PROGRAM IO_OP10_PANEL
VAR
	OP10_MP_16DI_MODULE_1 AT %I* : WORD;
	OP10_MP_16DI_MODULE_2 AT %I* : WORD;
	OP10_MP_16DI_MODULE_3 AT %I* : WORD;
	OP10_MP_16DI_MODULE_4 AT %I* : WORD;
	OP10_MP_16DI_MODULE_5 AT %I* : WORD;
	OP10_MP_16DI_MODULE_6 AT %I* : WORD;
	
	OP10_MP_16DO_MODULE_1 AT %Q* : WORD;
	OP10_MP_16DO_MODULE_2 AT %Q* : WORD;
	OP10_MP_16DO_MODULE_3 AT %Q* : WORD;
	OP10_MP_16DO_MODULE_4 AT %Q* : WORD;
	OP10_MP_16DO_MODULE_5 AT %Q* : WORD;
	
	WORD_AS_BIT_0: WORD_AS_BIT;
	WORD_AS_BIT_1: WORD_AS_BIT;
	WORD_AS_BIT_2: WORD_AS_BIT;
	WORD_AS_BIT_3: WORD_AS_BIT;
	WORD_AS_BIT_4: WORD_AS_BIT;
	WORD_AS_BIT_5: WORD_AS_BIT;

	BIT_AS_WORD_0: BIT_AS_WORD;
	BIT_AS_WORD_1: BIT_AS_WORD;
	BIT_AS_WORD_2: BIT_AS_WORD;
	BIT_AS_WORD_3: BIT_AS_WORD;
	BIT_AS_WORD_4: BIT_AS_WORD;
	OP10_MP_Spare_byte: WORD;
END_VAR

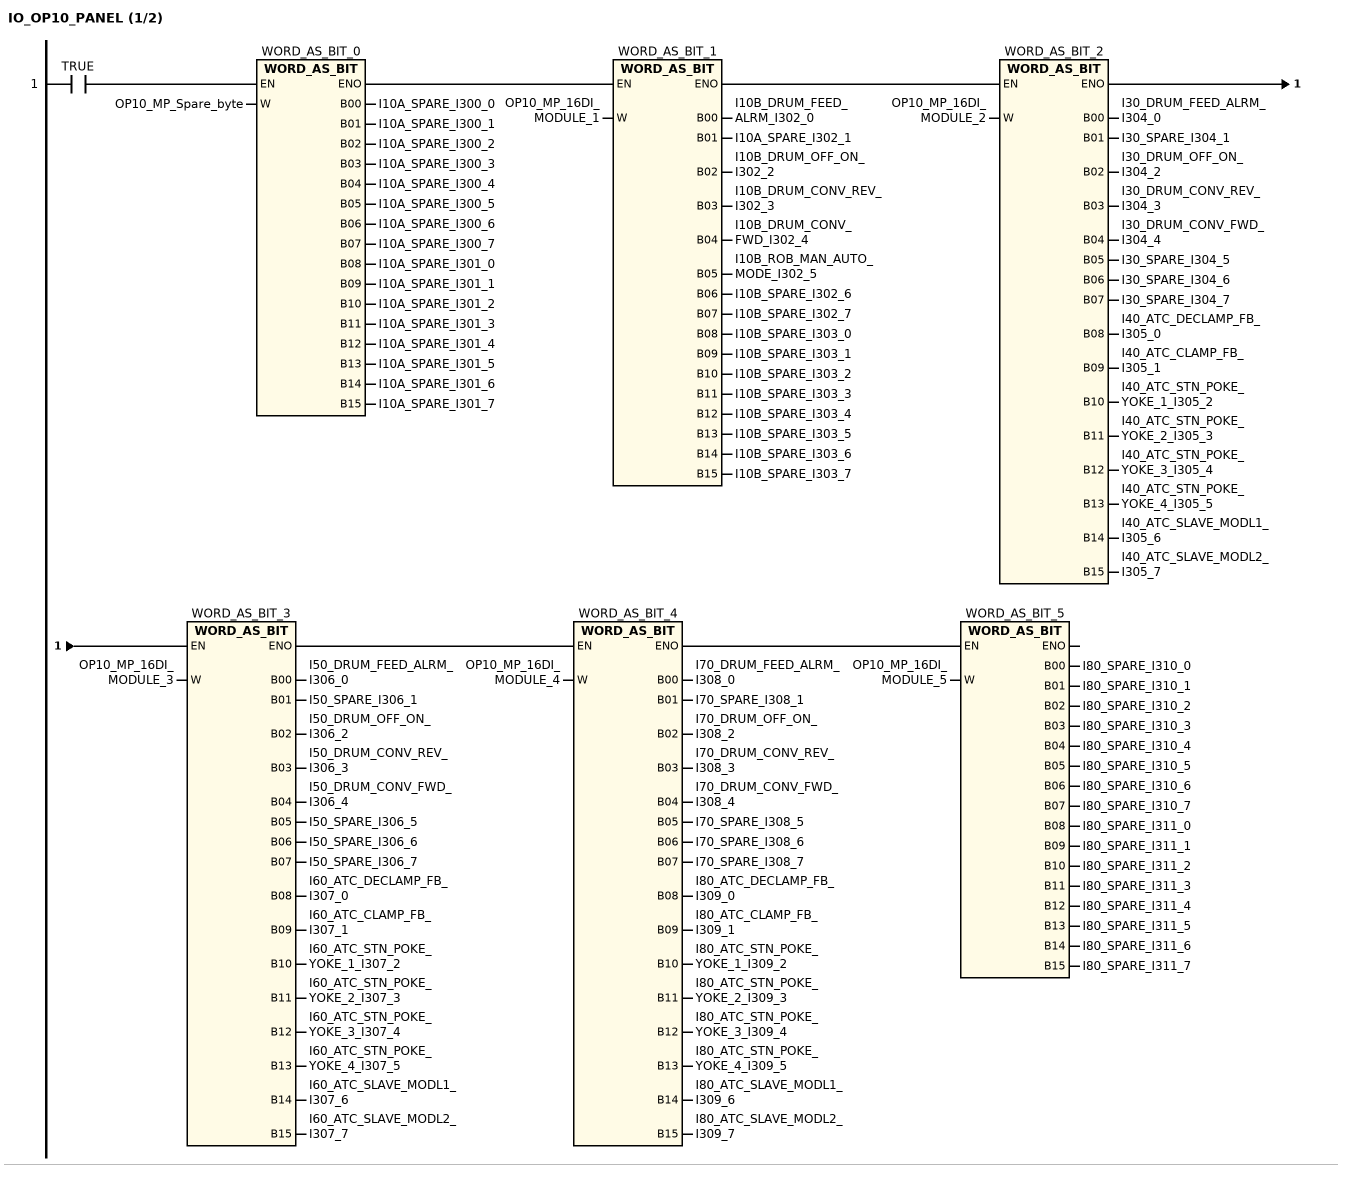
// NETWORK 1
WORD_AS_BIT_0(
    W := OP10_MP_Spare_byte,
    B00 => I10A_SPARE_I300_0,
    B01 => I10A_SPARE_I300_1,
    B02 => I10A_SPARE_I300_2,
    B03 => I10A_SPARE_I300_3,
    B04 => I10A_SPARE_I300_4,
    B05 => I10A_SPARE_I300_5,
    B06 => I10A_SPARE_I300_6,
    B07 => I10A_SPARE_I300_7,
    B08 => I10A_SPARE_I301_0,
    B09 => I10A_SPARE_I301_1,
    B10 => I10A_SPARE_I301_2,
    B11 => I10A_SPARE_I301_3,
    B12 => I10A_SPARE_I301_4,
    B13 => I10A_SPARE_I301_5,
    B14 => I10A_SPARE_I301_6,
    B15 => I10A_SPARE_I301_7); // WORD_AS_BIT
WORD_AS_BIT_1(
    W := OP10_MP_16DI_MODULE_1,
    B00 => I10B_DRUM_FEED_ALRM_I302_0,
    B01 => I10A_SPARE_I302_1,
    B02 => I10B_DRUM_OFF_ON_I302_2,
    B03 => I10B_DRUM_CONV_REV_I302_3,
    B04 => I10B_DRUM_CONV_FWD_I302_4,
    B05 => I10B_ROB_MAN_AUTO_MODE_I302_5,
    B06 => I10B_SPARE_I302_6,
    B07 => I10B_SPARE_I302_7,
    B08 => I10B_SPARE_I303_0,
    B09 => I10B_SPARE_I303_1,
    B10 => I10B_SPARE_I303_2,
    B11 => I10B_SPARE_I303_3,
    B12 => I10B_SPARE_I303_4,
    B13 => I10B_SPARE_I303_5,
    B14 => I10B_SPARE_I303_6,
    B15 => I10B_SPARE_I303_7); // WORD_AS_BIT
WORD_AS_BIT_2(
    W := OP10_MP_16DI_MODULE_2,
    B00 => I30_DRUM_FEED_ALRM_I304_0,
    B01 => I30_SPARE_I304_1,
    B02 => I30_DRUM_OFF_ON_I304_2,
    B03 => I30_DRUM_CONV_REV_I304_3,
    B04 => I30_DRUM_CONV_FWD_I304_4,
    B05 => I30_SPARE_I304_5,
    B06 => I30_SPARE_I304_6,
    B07 => I30_SPARE_I304_7,
    B08 => I40_ATC_DECLAMP_FB_I305_0,
    B09 => I40_ATC_CLAMP_FB_I305_1,
    B10 => I40_ATC_STN_POKE_YOKE_1_I305_2,
    B11 => I40_ATC_STN_POKE_YOKE_2_I305_3,
    B12 => I40_ATC_STN_POKE_YOKE_3_I305_4,
    B13 => I40_ATC_STN_POKE_YOKE_4_I305_5,
    B14 => I40_ATC_SLAVE_MODL1_I305_6,
    B15 => I40_ATC_SLAVE_MODL2_I305_7); // WORD_AS_BIT
WORD_AS_BIT_3(
    W := OP10_MP_16DI_MODULE_3,
    B00 => I50_DRUM_FEED_ALRM_I306_0,
    B01 => I50_SPARE_I306_1,
    B02 => I50_DRUM_OFF_ON_I306_2,
    B03 => I50_DRUM_CONV_REV_I306_3,
    B04 => I50_DRUM_CONV_FWD_I306_4,
    B05 => I50_SPARE_I306_5,
    B06 => I50_SPARE_I306_6,
    B07 => I50_SPARE_I306_7,
    B08 => I60_ATC_DECLAMP_FB_I307_0,
    B09 => I60_ATC_CLAMP_FB_I307_1,
    B10 => I60_ATC_STN_POKE_YOKE_1_I307_2,
    B11 => I60_ATC_STN_POKE_YOKE_2_I307_3,
    B12 => I60_ATC_STN_POKE_YOKE_3_I307_4,
    B13 => I60_ATC_STN_POKE_YOKE_4_I307_5,
    B14 => I60_ATC_SLAVE_MODL1_I307_6,
    B15 => I60_ATC_SLAVE_MODL2_I307_7); // WORD_AS_BIT
WORD_AS_BIT_4(
    W := OP10_MP_16DI_MODULE_4,
    B00 => I70_DRUM_FEED_ALRM_I308_0,
    B01 => I70_SPARE_I308_1,
    B02 => I70_DRUM_OFF_ON_I308_2,
    B03 => I70_DRUM_CONV_REV_I308_3,
    B04 => I70_DRUM_CONV_FWD_I308_4,
    B05 => I70_SPARE_I308_5,
    B06 => I70_SPARE_I308_6,
    B07 => I70_SPARE_I308_7,
    B08 => I80_ATC_DECLAMP_FB_I309_0,
    B09 => I80_ATC_CLAMP_FB_I309_1,
    B10 => I80_ATC_STN_POKE_YOKE_1_I309_2,
    B11 => I80_ATC_STN_POKE_YOKE_2_I309_3,
    B12 => I80_ATC_STN_POKE_YOKE_3_I309_4,
    B13 => I80_ATC_STN_POKE_YOKE_4_I309_5,
    B14 => I80_ATC_SLAVE_MODL1_I309_6,
    B15 => I80_ATC_SLAVE_MODL2_I309_7); // WORD_AS_BIT
WORD_AS_BIT_5(
    W := OP10_MP_16DI_MODULE_5,
    B00 => I80_SPARE_I310_0,
    B01 => I80_SPARE_I310_1,
    B02 => I80_SPARE_I310_2,
    B03 => I80_SPARE_I310_3,
    B04 => I80_SPARE_I310_4,
    B05 => I80_SPARE_I310_5,
    B06 => I80_SPARE_I310_6,
    B07 => I80_SPARE_I310_7,
    B08 => I80_SPARE_I311_0,
    B09 => I80_SPARE_I311_1,
    B10 => I80_SPARE_I311_2,
    B11 => I80_SPARE_I311_3,
    B12 => I80_SPARE_I311_4,
    B13 => I80_SPARE_I311_5,
    B14 => I80_SPARE_I311_6,
    B15 => I80_SPARE_I311_7); // WORD_AS_BIT

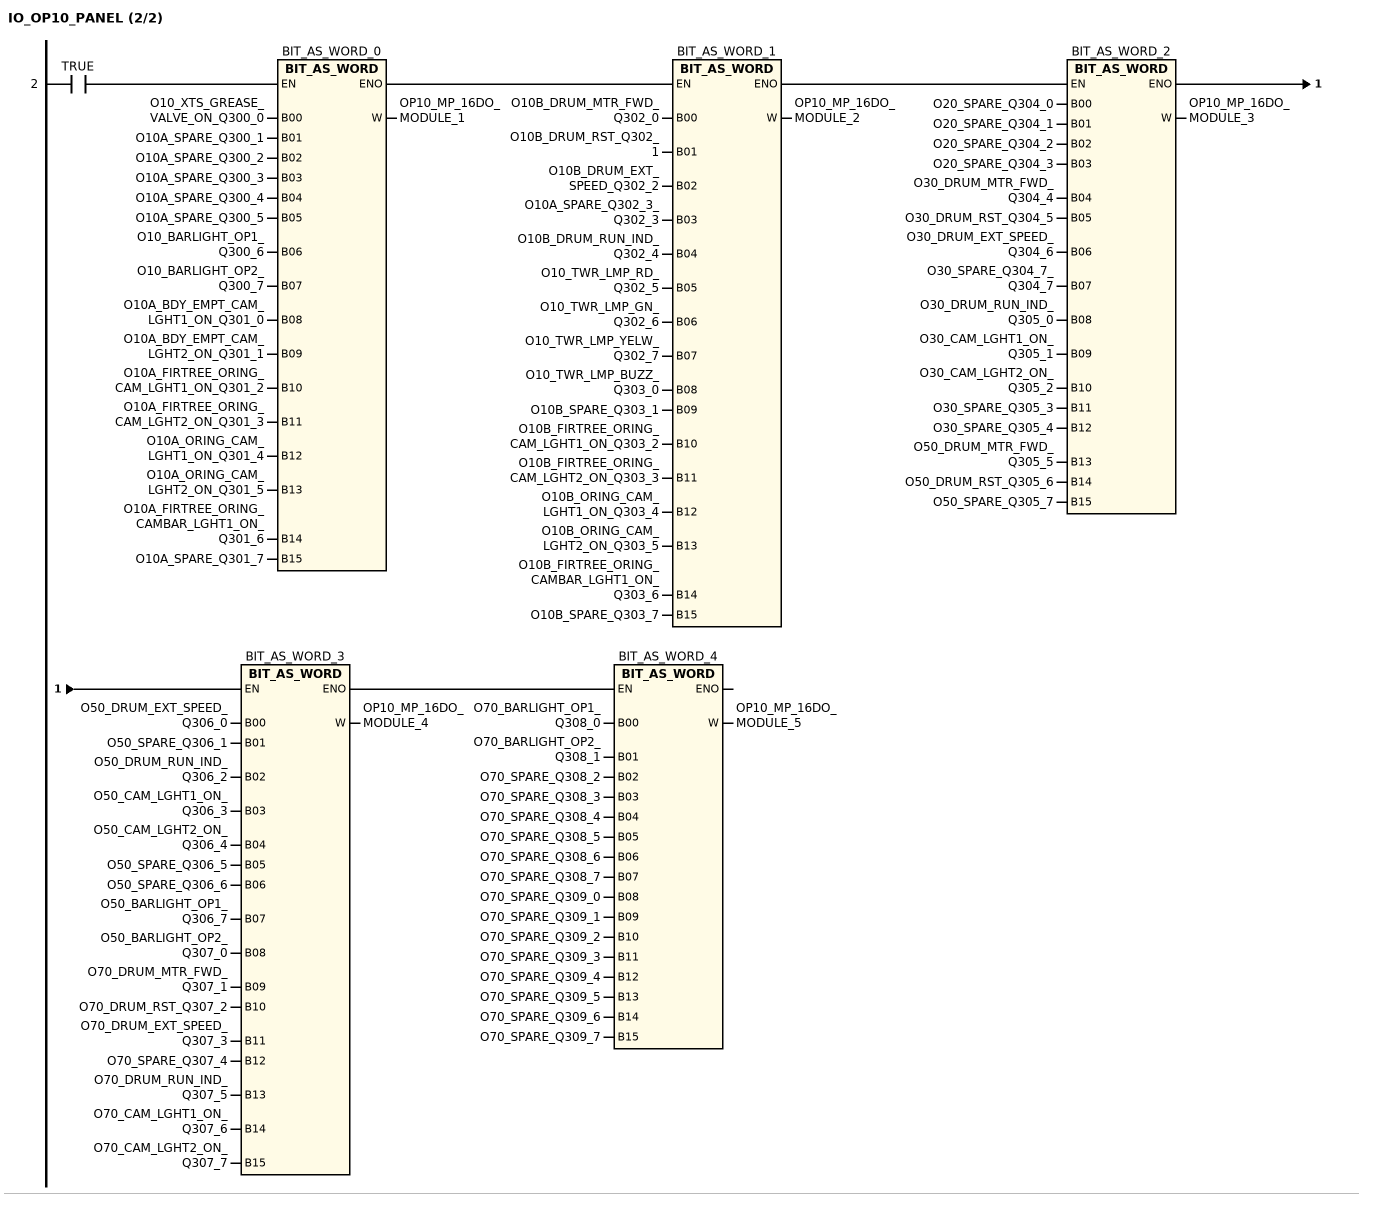
// NETWORK 2
BIT_AS_WORD_0(
    B00 := O10_XTS_GREASE_VALVE_ON_Q300_0,
    B01 := O10A_SPARE_Q300_1,
    B02 := O10A_SPARE_Q300_2,
    B03 := O10A_SPARE_Q300_3,
    B04 := O10A_SPARE_Q300_4,
    B05 := O10A_SPARE_Q300_5,
    B06 := O10_BARLIGHT_OP1_Q300_6,
    B07 := O10_BARLIGHT_OP2_Q300_7,
    B08 := O10A_BDY_EMPT_CAM_LGHT1_ON_Q301_0,
    B09 := O10A_BDY_EMPT_CAM_LGHT2_ON_Q301_1,
    B10 := O10A_FIRTREE_ORING_CAM_LGHT1_ON_Q301_2,
    B11 := O10A_FIRTREE_ORING_CAM_LGHT2_ON_Q301_3,
    B12 := O10A_ORING_CAM_LGHT1_ON_Q301_4,
    B13 := O10A_ORING_CAM_LGHT2_ON_Q301_5,
    B14 := O10A_FIRTREE_ORING_CAMBAR_LGHT1_ON_Q301_6,
    B15 := O10A_SPARE_Q301_7,
    W => OP10_MP_16DO_MODULE_1); // BIT_AS_WORD
BIT_AS_WORD_1(
    B00 := O10B_DRUM_MTR_FWD_Q302_0,
    B01 := O10B_DRUM_RST_Q302_1,
    B02 := O10B_DRUM_EXT_SPEED_Q302_2,
    B03 := O10A_SPARE_Q302_3_Q302_3,
    B04 := O10B_DRUM_RUN_IND_Q302_4,
    B05 := O10_TWR_LMP_RD_Q302_5,
    B06 := O10_TWR_LMP_GN_Q302_6,
    B07 := O10_TWR_LMP_YELW_Q302_7,
    B08 := O10_TWR_LMP_BUZZ_Q303_0,
    B09 := O10B_SPARE_Q303_1,
    B10 := O10B_FIRTREE_ORING_CAM_LGHT1_ON_Q303_2,
    B11 := O10B_FIRTREE_ORING_CAM_LGHT2_ON_Q303_3,
    B12 := O10B_ORING_CAM_LGHT1_ON_Q303_4,
    B13 := O10B_ORING_CAM_LGHT2_ON_Q303_5,
    B14 := O10B_FIRTREE_ORING_CAMBAR_LGHT1_ON_Q303_6,
    B15 := O10B_SPARE_Q303_7,
    W => OP10_MP_16DO_MODULE_2); // BIT_AS_WORD
BIT_AS_WORD_2(
    B00 := O20_SPARE_Q304_0,
    B01 := O20_SPARE_Q304_1,
    B02 := O20_SPARE_Q304_2,
    B03 := O20_SPARE_Q304_3,
    B04 := O30_DRUM_MTR_FWD_Q304_4,
    B05 := O30_DRUM_RST_Q304_5,
    B06 := O30_DRUM_EXT_SPEED_Q304_6,
    B07 := O30_SPARE_Q304_7_Q304_7,
    B08 := O30_DRUM_RUN_IND_Q305_0,
    B09 := O30_CAM_LGHT1_ON_Q305_1,
    B10 := O30_CAM_LGHT2_ON_Q305_2,
    B11 := O30_SPARE_Q305_3,
    B12 := O30_SPARE_Q305_4,
    B13 := O50_DRUM_MTR_FWD_Q305_5,
    B14 := O50_DRUM_RST_Q305_6,
    B15 := O50_SPARE_Q305_7,
    W => OP10_MP_16DO_MODULE_3); // BIT_AS_WORD
BIT_AS_WORD_3(
    B00 := O50_DRUM_EXT_SPEED_Q306_0,
    B01 := O50_SPARE_Q306_1,
    B02 := O50_DRUM_RUN_IND_Q306_2,
    B03 := O50_CAM_LGHT1_ON_Q306_3,
    B04 := O50_CAM_LGHT2_ON_Q306_4,
    B05 := O50_SPARE_Q306_5,
    B06 := O50_SPARE_Q306_6,
    B07 := O50_BARLIGHT_OP1_Q306_7,
    B08 := O50_BARLIGHT_OP2_Q307_0,
    B09 := O70_DRUM_MTR_FWD_Q307_1,
    B10 := O70_DRUM_RST_Q307_2,
    B11 := O70_DRUM_EXT_SPEED_Q307_3,
    B12 := O70_SPARE_Q307_4,
    B13 := O70_DRUM_RUN_IND_Q307_5,
    B14 := O70_CAM_LGHT1_ON_Q307_6,
    B15 := O70_CAM_LGHT2_ON_Q307_7,
    W => OP10_MP_16DO_MODULE_4); // BIT_AS_WORD
BIT_AS_WORD_4(
    B00 := O70_BARLIGHT_OP1_Q308_0,
    B01 := O70_BARLIGHT_OP2_Q308_1,
    B02 := O70_SPARE_Q308_2,
    B03 := O70_SPARE_Q308_3,
    B04 := O70_SPARE_Q308_4,
    B05 := O70_SPARE_Q308_5,
    B06 := O70_SPARE_Q308_6,
    B07 := O70_SPARE_Q308_7,
    B08 := O70_SPARE_Q309_0,
    B09 := O70_SPARE_Q309_1,
    B10 := O70_SPARE_Q309_2,
    B11 := O70_SPARE_Q309_3,
    B12 := O70_SPARE_Q309_4,
    B13 := O70_SPARE_Q309_5,
    B14 := O70_SPARE_Q309_6,
    B15 := O70_SPARE_Q309_7,
    W => OP10_MP_16DO_MODULE_5); // BIT_AS_WORD

END_PROGRAM

(* stored: Version 1.1.0.1, ProductVersion 3.1.4024.11
   POU IO_OP10_PANEL: Id {2e2f4e82-5379-4198-ace1-af53950ccc1b}, SpecialFunc None *)
